// LS Electric XG5000 project: 편솔1
// PLC LSPLC

PROGRAM NewProgram (task: 스캔 프로그램)

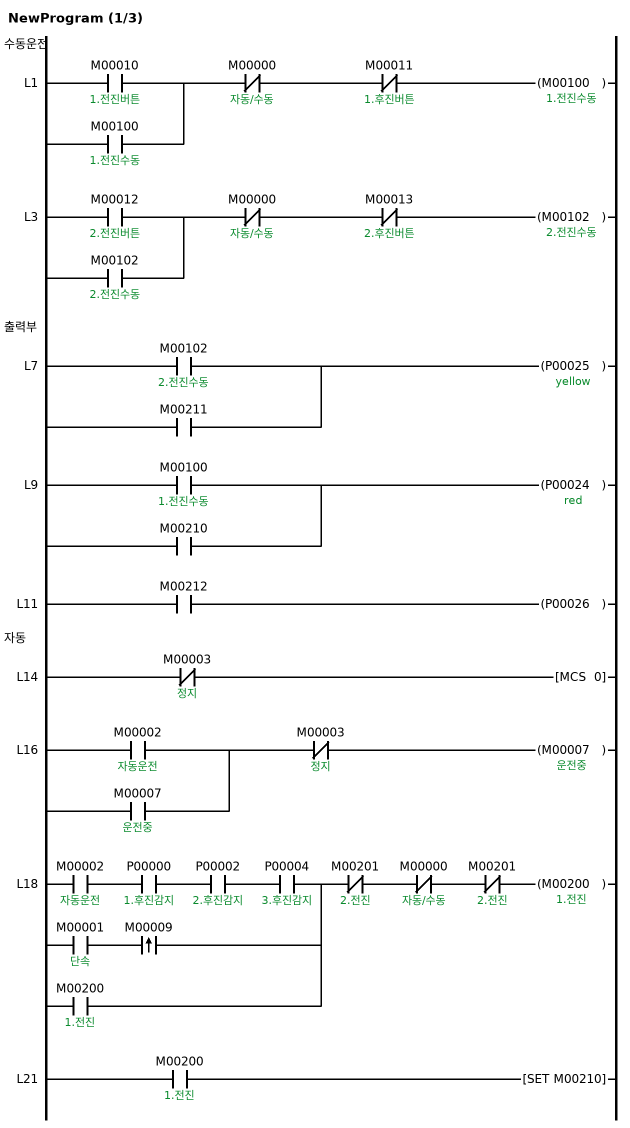
수동운전:
; L1
LOAD      M00010	// 1.전진버튼
OR        M00100	// 1.전진수동
AND NOT   M00000	// 자동/수동
AND NOT   M00011	// 1.후진버튼
OUT       M00100	// 1.전진수동
; L3
LOAD      M00012	// 2.전진버튼
OR        M00102	// 2.전진수동
AND NOT   M00000	// 자동/수동
AND NOT   M00013	// 2.후진버튼
OUT       M00102	// 2.전진수동
출력부:
; L7
LOAD      M00102	// 2.전진수동
OR        M00211
OUT       P00025	// yellow
; L9
LOAD      M00100	// 1.전진수동
OR        M00210
OUT       P00024	// red
; L11
LOAD      M00212
OUT       P00026
자동:
; L14
LOAD NOT  M00003	// 정지
MCS       0
; L16
LOAD      M00002	// 자동운전
OR        M00007	// 운전중
AND NOT   M00003	// 정지
OUT       M00007	// 운전중
; L18
LOAD      M00002	// 자동운전
AND       P00000	// 1.후진감지
AND       P00002	// 2.후진감지
AND       P00004	// 3.후진감지
LOAD      M00001	// 단속
ANDP      M00009
OR LOAD
OR        M00200	// 1.전진
AND NOT   M00201	// 2.전진
AND NOT   M00000	// 자동/수동
AND NOT   M00201	// 2.전진
OUT       M00200	// 1.전진
; L21
LOAD      M00200	// 1.전진
SET       M00210

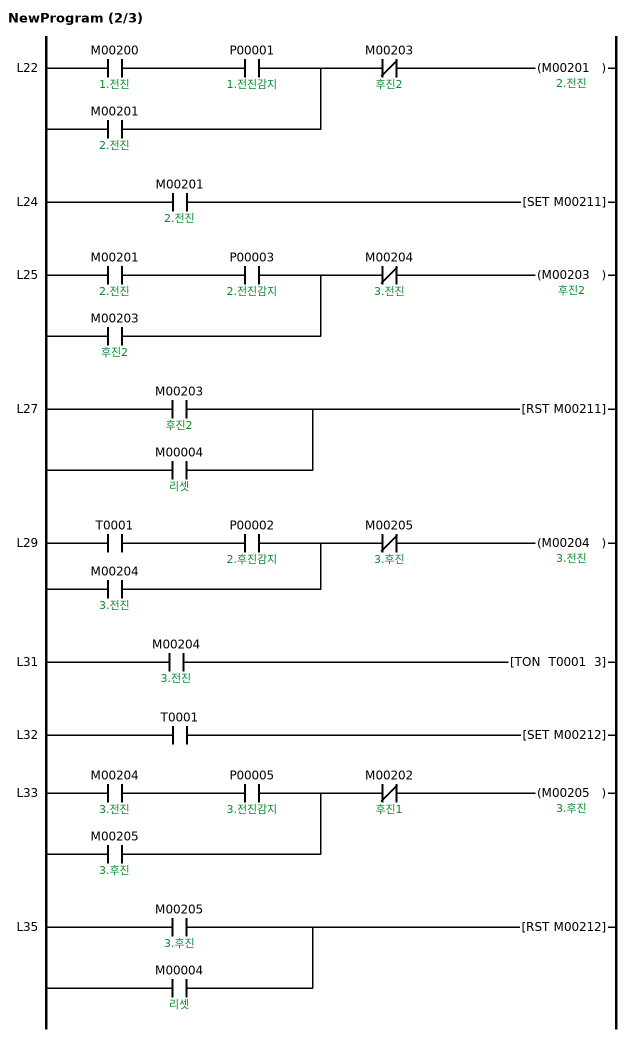
; L22
LOAD      M00200	// 1.전진
AND       P00001	// 1.전진감지
OR        M00201	// 2.전진
AND NOT   M00203	// 후진2
OUT       M00201	// 2.전진
; L24
LOAD      M00201	// 2.전진
SET       M00211
; L25
LOAD      M00201	// 2.전진
AND       P00003	// 2.전진감지
OR        M00203	// 후진2
AND NOT   M00204	// 3.전진
OUT       M00203	// 후진2
; L27
LOAD      M00203	// 후진2
OR        M00004	// 리셋
RST       M00211
; L29
LOAD      T0001
AND       P00002	// 2.후진감지
OR        M00204	// 3.전진
AND NOT   M00205	// 3.후진
OUT       M00204	// 3.전진
; L31
LOAD      M00204	// 3.전진
TON       T0001 3
; L32
LOAD      T0001
SET       M00212
; L33
LOAD      M00204	// 3.전진
AND       P00005	// 3.전진감지
OR        M00205	// 3.후진
AND NOT   M00202	// 후진1
OUT       M00205	// 3.후진
; L35
LOAD      M00205	// 3.후진
OR        M00004	// 리셋
RST       M00212

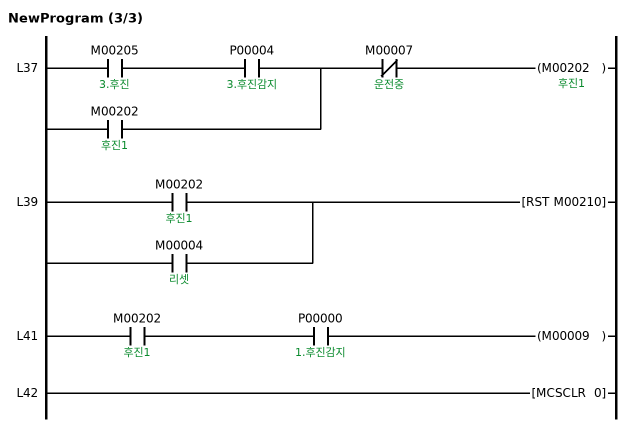
; L37
LOAD      M00205	// 3.후진
AND       P00004	// 3.후진감지
OR        M00202	// 후진1
AND NOT   M00007	// 운전중
OUT       M00202	// 후진1
; L39
LOAD      M00202	// 후진1
OR        M00004	// 리셋
RST       M00210
; L41
LOAD      M00202	// 후진1
AND       P00000	// 1.후진감지
OUT       M00009
; L42
MCSCLR    0

VARIABLES AND COMMENTS (devices not used above)
M00101	BIT	1.후진수동
M00103	BIT	2.후진수동
M00014	BIT	3.전진
M00015	BIT	3.후진
P00007	BIT	운정중